TYPE ST_HmiStatus :
STRUCT
    eMachineState             	: E_MachineState;
    eIndexState               	: E_IndexState;
    eIndexPosition           	: E_TablePosition;
	iPowerCountdown 		  	: INT := 0;
    iNestRotationAngle        	: INT;
    bReady                    	: BOOL;
    bBusy                     	: BOOL;
    bFaulted                  	: BOOL;
    bTwoHandsSafe             	: BOOL;
    bLoadingStationEaglePresent : BOOL;
    bRejectChutePartPresent   	: BOOL;
    bHeatStakeEaglePresent    	: BOOL;
    bHeatStakePatchPresent    	: BOOL;
    bPbupMagnetPresent        	: BOOL;
    bIndexReady               	: BOOL;
    bIndexLocked              	: BOOL;
    bIndexCompletedSensor     	: BOOL;
    bMainDoorClosed           	: BOOL;
    bMainDoorLocked           	: BOOL;
    bStartButtonActive        	: BOOL;
    bStopButtonActive         	: BOOL;
    bResetButtonActive        	: BOOL;
    bStartButtonLamp          	: BOOL;
    bUp24VPowerSupplyOk       	: BOOL;
    bUs24VPowerSupplyOk       	: BOOL;
    b48VPowerSupplyOk         	: BOOL;
    bMainDoorDiagnosticOk     	: BOOL;
    bMs6FeedbackOk            	: BOOL;
    bAirExhausted             	: BOOL;
    bLeftFlapSafe             	: BOOL;
    bRightFlapSafe            	: BOOL;
    bEnableSettings           	: BOOL;
    bAllStationsCommissioned  	: BOOL;
    bAutoCycleAllowed         	: BOOL;

    bNest1Blocked             			: BOOL;
    bNest2Blocked             			: BOOL;
    bNest3Blocked             			: BOOL;
    bNest4Blocked             			: BOOL;

    bDisabledNestPartIndexBlocked 		: BOOL;
    bDisabledNestPartPopupRequest 		: BOOL;
    uiDisabledNestPartPopupNestId 		: UINT;
    sDisabledNestPartPopupMessage 		: STRING(255);

    // Reject chute full / controlled-stop status.
    bRejectChuteFullLatched   			: BOOL;
    bRejectChutePopupRequest 			: BOOL;
	bReprocessPopupRequest 				: BOOL;
    bRejectChuteStopRequest 			: BOOL;
    bRejectChuteResetBlocked 			: BOOL;
    sRejectChutePopupMessage 			: STRING(255);
	
	// Patch Dispensing Station - Nest Support
	bPatchSupportRetracted 				: BOOL;
	bPatchSupportExtended  				: BOOL;

    // Heat Stake head cylinder diagnostics.
    bHeatStakeHeadUp 					: BOOL;
    bHeatStakeHeadDown 					: BOOL;
    bHeatStakeHeadDownTimeoutFault 		: BOOL;
    bHeatStakeHeadUpTimeoutFault 		: BOOL;
    bHeatStakeHeadSensorConflictFault 	: BOOL;
	
	// =====================================================
	// Vision Manual Mode
	// =====================================================
	
	// General manual control
	bVisionManualEnableAllowed 			: BOOL;
	
	// Individual motion permissives
	bVisionHorizontalBackAllowed       	: BOOL;
	bVisionHorizontalFrontAllowed      	: BOOL;
	
	bVisionVerticalUpAllowed           	: BOOL;
	bVisionVerticalIntermediateAllowed 	: BOOL;
	bVisionVerticalFullDownAllowed     	: BOOL;
	
	bVisionGripOpenAllowed             	: BOOL;
	bVisionGripCloseAllowed            	: BOOL;
	
	bVisionRotate0Allowed              	: BOOL;
	bVisionRotate180Allowed            	: BOOL;
	
	bVisionSupportAllowed              	: BOOL;
	
	// Position feedback
	bVisionHorizontalBack  				: BOOL;
	bVisionHorizontalFront 				: BOOL;
	
	bVisionVerticalUp      				: BOOL;
	bVisionVerticalDown    				: BOOL;
	
	bVisionGripOpen        				: BOOL;
	bVisionGripClosed      				: BOOL;
	
	bVisionRotate0         				: BOOL;
	bVisionRotate180       				: BOOL;
	
	bVisionSupportExtended  			: BOOL;
	bVisionSupportRetracted 			: BOOL;

    stPatchDispense           			: ST_PatchStageStatus;
    stHeatStake               			: ST_PatchStageStatus;
    stHeatStakeTemperature    			: ST_HeatStakeTemperatureStatus;
    stHeatStakeProcess        			: ST_HeatStakeProcessStatus;
    stHeatStakeProcessSettings 			: ST_HeatStakeProcessSettings;
    bHeatStakeProcessSettingsWriteBusy 	: BOOL;
    bHeatStakeProcessSettingsWriteError : BOOL;
    udiHeatStakeProcessSettingsWriteErrorId : UDINT;
    stHeatStakeTemperatureSettings 		: ST_HeatStakeTemperatureSettings;
    bHeatStakeSettingsApplyAccepted 	: BOOL;
    bHeatStakeSettingsApplyRejected 	: BOOL;
    bHeatStakeSettingsWriteBusy 		: BOOL;
    bHeatStakeSettingsWriteError 		: BOOL;
    bHeatStakeSettingsSaveSuccessful 	: BOOL;
    bHeatStakeSettingsSaveFailed 		: BOOL;
    sHeatStakeSettingsApplyRejectReason : STRING(255);
    udiHeatStakeSettingsWriteErrorId 	: UDINT;

    // Current physical nest at each process station.
    uiPatchDispenseNestId 				: UINT;
    uiHeatStakeNestId     				: UINT;
    uiVisionNestId        				: UINT;

    bHeatStakeManualEnableAllowed     	: BOOL;
    bHeatStakeManualStakeAllowed      	: BOOL;
    bHeatStakeManualUnlockAllowed     	: BOOL;
    bHeatStakeManualLockAllowed       	: BOOL;
    bHeatStakeManualHeadDownAllowed   	: BOOL;
    bHeatStakeManualHeadUpAllowed     	: BOOL;
    bHeatStakeManualSupportAllowed    	: BOOL;
    bHeatStakeManualActionBusy        	: BOOL;
    bHeatStakeManualHeadUnlocked      	: BOOL;
	bVisionManualRunSequenceAllowed   	: BOOL;
	bVisionManualHomeAllowed 		 	: BOOL;
	bVisionHome              		  	: BOOL;

    stVision                  			: ST_PatchStageStatus;
    eOperatorInstruction      			: E_OperatorInstruction;
    stOperatorStation         			: ST_OperatorStationStatus;
    aNest                     			: ARRAY[1..4] OF ST_Nest;
    sMachineMessage           			: STRING(160);
    sOperatorMessage          			: STRING(255);
    sAutoCycleBlockReason     			: STRING(160);
	
	
    bLoadingStationPbupPresent : BOOL; // Operator PBUP sensor; provisional Term19 Input1
END_STRUCT
END_TYPE

(* stored: Version 1.1.0.1, ProductVersion 3.1.4026.18
   DUT ST_HmiStatus: Id {d41f7c8f-993e-495c-ab35-890ed277e5d6} *)
